PROGRAM PRG_ShutdownPLC
VAR
	fbReboot    : NT_Reboot;
    fbShutdown  : NT_Shutdown;
    fbWritePersistentData : FB_WritePersistentData;

    fbR_Trig        	: R_TRIG;
    tonSafeShutdown   	: TON;
    tonSafeReboot     	: TON;
	tonPowerSupplyDelay	: TON;

    bStart              : BOOL := TRUE;
    bWriteDone          : BOOL := FALSE;
    bShutdownRequest    : BOOL := FALSE;
    bRebootRequest      : BOOL := FALSE;
	bPowerSupplyDelay	: BOOL := FALSE;
	
	tRebootTime		: TIME := T#10S;
	tShutdownTime	: TIME := T#60S;
	
END_VAR

// === Check if power supply is NOT OK or Shutdown is requested by HMI ===
tonPowerSupplyDelay( IN := bPowerSupplyDelay, PT := T#3S);

bPowerSupplyDelay := NOT (GVL_IO.gDigInputs.b24VPowerSupplyOK AND GVL_IO.gDigInputs.b24VPowerSupplyOKBck AND GVL_IO.gDigInputs.b48VPowerSupplyOK AND GVL_IO.gDigInputs.b48VPowerSupplyOKBck);

IF tonPowerSupplyDelay.Q OR GVL_HMI.HMIDigInputs.bShutdownPLC THEN

    // === Trigger on rising edge of START to prevent multiple writes ===
    fbR_Trig(CLK := bStart);

    IF fbR_Trig.Q THEN
        // Start writing RETAIN/PERSISTENT variables to non-volatile memory
        fbWritePersistentData(NETID := '', PORT := 851, START := TRUE, TMOUT := T#1s);
    ELSE
        fbWritePersistentData(START := FALSE);
    END_IF

    // === Start Shutdown Timer only after successful write ===
    IF NOT fbWritePersistentData.BUSY AND NOT fbWritePersistentData.ERR THEN
        bWriteDone := TRUE;
    END_IF

    IF bWriteDone THEN
        tonSafeShutdown(IN := TRUE, PT := tShutdownTime);
		GVL_HMI.rTimeCountingDown   := (TIME_TO_DWORD(tShutdownTime)/1000) - (TIME_TO_DWORD(tonSafeShutdown.ET)/1000);
		GVL_HMI.sCountdownPopupText := 'Shutdown';
    END_IF
ELSE
    // Reset shutdown timer and write flag if no shutdown condition
    tonSafeShutdown(IN := FALSE);
    bWriteDone := FALSE;
	
END_IF


// === Check if Reboot command from HMI is active ===
IF GVL_HMI.HMIDigInputs.bRebootPLC THEN
    tonSafeReboot(IN := TRUE, PT := T#10S);
	GVL_HMI.rTimeCountingDown := 10 - TIME_TO_DWORD(tonSafeReboot.ET)/1000;
	GVL_HMI.sCountdownPopupText := 'Reboot';
ELSE
    tonSafeReboot(IN := FALSE);
END_IF


// === After timers expire, set action flags ===
IF tonSafeShutdown.Q THEN
    bShutdownRequest := TRUE;
END_IF

IF tonSafeReboot.Q THEN
    bRebootRequest := TRUE;
END_IF


// === Execute Reboot ===
fbReboot(Start := bRebootRequest);

// === Execute Shutdown ===
fbShutdown(Start := bShutdownRequest);

END_PROGRAM

(* stored: Version 1.1.0.1, ProductVersion 3.1.4024.15
   POU PRG_ShutdownPLC: Id {71ae888e-9b37-420e-9d56-8353899fcb8d}, SpecialFunc None *)
